Fanuc KAREL source: kt00439.KL

-- PROVISIONAL review KL for V940-1; original PC SHA256 01cb9ce9cf16def7d923ab1a68dfdad2e5c8d51c736bcf231b0894e25a18c52a
-- Incomplete behavior may be omitted. Consult companion uncertainty JSON. Do not deploy.
PROGRAM KT00439
%NOLOCKGROUP
VAR
  I1 : INTEGER
  OUT : BOOLEAN
-- UNRESOLVED_DECL Y2 type=002018
BEGIN
  -- V9_ZERO_TABLE_METADATA_HINT layout=0001; no indexed target words; source/name/runtime held
  -- UNRESOLVED_PC offsets 5-16; opcodes 2E,23
  -- UNRESOLVED_PC offsets 21-35; opcodes 2E,22,9D,33,B2
  -- UNRESOLVED_PC offsets 40-62; opcodes 21,22,9D,33,B1,5C,23
  -- UNRESOLVED_PC offsets 67-71; opcodes 7F
END KT00439
